// TIA Portal V20 export
ORGANIZATION_BLOCK "Startup"   // OB100, SCL, Startup
TITLE = "Complete Restart"
{ S7_Optimized_Access := 'TRUE' }
// stored: SetENOAutomatically false
   VAR_INPUT
      LostRetentive : Bool;   // True if retentive data are lost
      LostRTC : Bool;   // True if date and time are lost
   END_VAR
   VAR_TEMP
      tLastDateTime : DTL;
      tLasDateTimeSec : DInt;
      tActualDateTime : DTL;
      tActualDateTimeINT : DInt;
      tActualDateTimeSec : DInt;
   END_VAR
BEGIN
   REGION Description head
       //==================================================================================
       // POSALUX Swiss SA / (C) Copyright 2025
       //----------------------------------------------------------------------------------
       // Title: Startup
       // Comment/Function: Executes one time when the operating mode of the CPU changes from STOP to RUN
       // Author: Fabien WALDT
       // Engineering: TIA Portal v19
       //----------------------------------------------------------------------------------
       // Change log table:
       // Version  | Date     | Expert in charge | Changes applied
       //----------------------------------------------------------------------------------
       // 00.00.01 | 20250423 | WFA              | First released version
       //==================================================================================
   END_REGION

   REGION Safety Brake Test
       "LBP_AlarmMsgs".UserA[5].A70UUxx[12] := FALSE;  // Msg 700512 "SAFETY : THE BRAKE TEST IS NOT WORKING, PLEASE RESET"
   END_REGION

   REGION Config NC Panel
       "LBP_ConfigBP"(MCPNum := "LBP_ConfigData".MCPNum,
                      MCP1In := "MCP1_In",
                      MCP1Out := "MCP1_Out",
                      MCP1BusAdr := "LBP_ConfigData".MCP1BusAdr,
                      MCP1Timeout := "LBP_ConfigData".MCP1Timeout,
                      MCP2In := NULL,
                      MCP2Out := NULL,
                      MCP2BusAdr := "LBP_ConfigData".MCP2BusAdr,
                      MCP2Timeout := "LBP_ConfigData".MCP2Timeout,
                      MCP1Stop := "LBP_ConfigData".MCP1Stop,
                      MCP2Stop := "LBP_ConfigData".MCP2Stop,
                      MCP1NotSend := "LBP_ConfigData".MCP1NotSend,
                      MCP2NotSend := "LBP_ConfigData".MCP2NotSend,
                      MCPBusType := "LBP_ConfigData".MCPBusType,
                      HTIf := "LBP_ConfigData".HTIf,
                      HTIn := "LBP_ConfigData".HTIn,
                      HTOut := "LBP_ConfigData".HTOut,
                      HTAdr := "LBP_ConfigData".HTAdr,
                      HTStop := "LBP_ConfigData".HTStop,
                      HTNotSend := "LBP_ConfigData".HTNotSend,
                      NCCyclTimeout := "LBP_ConfigData".NCCyclTimeout,
                      NCRunupTimeout := "LBP_ConfigData".NCRunupTimeout,
                      ListMDecGrp := "LBP_ConfigData".ListMDecGrp,
                      MMCToIF := "LBP_ConfigData".MMCToIF,
                      HWheelMMC := "LBP_ConfigData".HWheelMMC,
                      MCP_IF_TCS := "LBP_ConfigData".MCP_IF_TCS,
                      ExtendChanAxMsg := "LBP_ConfigData".ExtendChanAxMsg,
                      HMIAxisSel := "LBP_ConfigData".HMIAxisSel,
                      DeactivateCtrlEnergy:=FALSE,
                      MsgUser := "LBP_ConfigData".MsgUser,
                      IRAuxfuT := "LBP_ConfigData".IRAuxfuT,
                      IRAuxfuH := "LBP_ConfigData".IRAuxfuH,
                      IRAuxfuE := "LBP_ConfigData".IRAuxfuE,
                      UserVersion := "LBP_ConfigData".UserVersionInfo,
                      OpKeyNum := "LBP_ConfigData".OpKeyNum,
                      Op1KeyIn := "LBP_ConfigData".Op1KeyIn,
                      Op1KeyOut := "LBP_ConfigData".Op1KeyOut,
                      Op1KeyBusAdr := "LBP_ConfigData".Op1KeyBusAdr,
                      Op2KeyIn := "LBP_ConfigData".Op2KeyIn,
                      Op2KeyOut := "LBP_ConfigData".Op2KeyOut,
                      Op2KeyBusAdr := "LBP_ConfigData".Op2KeyBusAdr,
                      Op1KeyStop := "LBP_ConfigData".Op1KeyStop,
                      Op2KeyStop := "LBP_ConfigData".Op2KeyStop,
                      Op1KeyNotSend := "LBP_ConfigData".Op1KeyNotSend,
                      Op2KeyNotSend := "LBP_ConfigData".Op2KeyNotSend,
                      OpUnitCommId := "LBP_ConfigData".OpUnitCommId,
                      OpUnitInterfaceId := "LBP_ConfigData".OpUnitInterfaceId,
                      MCP1ConnectionId := "LBP_ConfigData".MCP1ConnectionId,
                      MCP2ConnectionId := "LBP_ConfigData".MCP2ConnectionId,
                      HTConnectionId := "LBP_ConfigData".HTConnectionId,
                      Op1KeyConnectionId := "LBP_ConfigData".Op1KeyConnectionId,
                      Op2KeyConnectionId := "LBP_ConfigData".Op2KeyConnectionId,
                      IdentConnectionId := "LBP_ConfigData".IdentConnectionId,
                      MCP1LocalUdpPort := "LBP_ConfigData".MCP1LocalUdpPort,
                      MCP2LocalUdpPort := "LBP_ConfigData".MCP2LocalUdpPort,
                      HTLocalUdpPort := "LBP_ConfigData".HTLocalUdpPort,
                      Op1KeyLocalUdpPort := "LBP_ConfigData".Op1KeyLocalUdpPort,
                      Op2KeyLocalUdpPort := "LBP_ConfigData".Op2KeyLocalUdpPort,
                      IdentLocalUdpPort := "LBP_ConfigData".IdentLocalUdpPort,
                      MaxModeGroup => "LBP_ConfigData".MaxModeGroup,
                      MaxChan => "LBP_ConfigData".MaxChan,
                      MaxAxis => "LBP_ConfigData".MaxAxis,
                      ActiveChan => "LBP_ConfigData".ActiveChan,
                      ActiveAxis => "LBP_ConfigData".ActiveAxis,
                      MaxNumUserDataInt => "LBP_ConfigData".MaxNumUserDataInt,
                      MaxNumUserDataHex => "LBP_ConfigData".MaxNumUserDataHex,
                      MaxNumUserDataReal => "LBP_ConfigData".MaxNumUserDataReal,
                      UserDataIntArray => NULL,
                      UserDataHexArray => NULL,
                      UserDataRealArray => NULL,
                      TMMagazines => NULL);
   END_REGION

   REGION RAZ Shutdown variables
       "LBP_AlarmMsgs".UserA[04].A70UUxx[05] := FALSE;  // Msg 700405 "UPS power failure"
       "LBP_AlarmMsgs".UserA[04].A70UUxx[41] := FALSE;  // Msg 700441 "Machine stop process completed. Turn off the machine using the main switch"
       "LBP_AlarmMsgs".UserA[04].A70UUxx[42] := FALSE;  // Msg 700442 "The machine stop process has started..."
       "LBP_AlarmMsgs".UserA[04].A70UUxx[20] := FALSE;  // Msg 700420 "Timeout shutdown. Please turn off manually"
       "LBP_AlarmMsgs".UserA[04].A70UUxx[21] := FALSE;  // Msg 700421 "The laser is still on. Please turn it off manually"
       "LBP_AlarmMsgs".UserA[04].A70UUxx[22] := FALSE;  // Msg 700422 "Laser status unknown. Turn it off on left PC then wait for the machine's shutdown"
       "LBP_AlarmMsgs".UserA[04].A70UUxx[23] := FALSE;  // Msg 700423 "Power failure. The machine stop process has started…"

       "DB_Machineshutdown_UPS".sShutDownPCRequest    := 0;
       "DB_Machineshutdown_UPS".sShutDownPCResponse   := 0;
   END_REGION
END_ORGANIZATION_BLOCK
